// TIA Portal V20 export
DATA_BLOCK "InstStackCalculateDB"   // DB459
// stored: InstanceOfName 2201_StackCalculate, InstanceOfType FB
"2201_StackCalculate"
   // VAR_INPUT
   //    Execute : Bool;
   //    Direction : Bool;
   //    CPM : LReal;
   //    StageWidth : LReal;
   //    StageHeight : LReal;
   //    StageGap : LReal;
   //    AccRatio : DInt;
   //    RatioOption : Bool;
   //    TimeOption : Bool;
   //    PosOption : Bool;
   //    DoubleOption : Bool;
   //    Ratio : Struct
   //       FinalRollerStart : LReal;
   //       FinalRollerEnd : LReal;
   //       PnPXStart : LReal;
   //       PnPXEnd : LReal;
   //       PnPZDownStart : LReal;
   //       PnPZDownEnd : LReal;
   //       PnPZUpStart : LReal;
   //       PnPZUpEnd : LReal;
   //       MandrelBwdStart : LReal;
   //       MandrelBwdEnd : LReal;
   //       MandrelFwdStart : LReal;
   //       MandrelFwdEnd : LReal;
   //       MandrelUpStart1 : LReal;
   //       MandrelUpEnd1 : LReal;
   //       MandrelUpStart2 : LReal;
   //       MandrelUpEnd2 : LReal;
   //       MandrelDownStart : LReal;
   //       MandrelDownEnd : LReal;
   //       MandrelYTerm : LReal;
   //       MandrelZTerm : LReal;
   //       MandrelBwdOffset : LReal;
   //       MandrelFwdOffset : LReal;
   //    END_STRUCT;
   //    "Time" : Struct
   //       FinalRollerStart : LReal;
   //       FinalRollerEnd : LReal;
   //       PnPXStart : LReal;
   //       PnPXEnd : LReal;
   //       PnPZDownStart : LReal;
   //       PnPZDownEnd : LReal;
   //       PnPZUpStart : LReal;
   //       PnPZUpEnd : LReal;
   //       MandrelBwdStart : LReal;
   //       MandrelBwdEnd : LReal;
   //       MandrelFwdStart : LReal;
   //       MandrelFwdEnd : LReal;
   //       MandrelUpStart1 : LReal;
   //       MandrelUpEnd1 : LReal;
   //       MandrelUpStart2 : LReal;
   //       MandrelUpEnd2 : LReal;
   //       MandrelDownStart : LReal;
   //       MandrelDownEnd : LReal;
   //    END_STRUCT;
   //    Position : Struct
   //       FinalRollerBwdPos : LReal;
   //       FinalRollerFwdPos : LReal;
   //    END_STRUCT;
   //    FinalRollerDistance : LReal;
   //    AnodePnPX1Distance : LReal;
   //    AnodePnPX2Distance : LReal;
   //    CathodePnPX1Distance : LReal;
   //    CathodePnPX2Distance : LReal;
   //    AnodePnPZ1Distance1 : LReal;
   //    AnodePnPZ1Distance2 : LReal;
   //    AnodePnPZ2Distance1 : LReal;
   //    AnodePnPZ2Distance2 : LReal;
   //    CathodePnPZ1Distance1 : LReal;
   //    CathodePnPZ1Distance2 : LReal;
   //    CathodePnPZ2Distance1 : LReal;
   //    CathodePnPZ2Distance2 : LReal;
   //    AnodeMandrelYFrontDistance : LReal;
   //    AnodeMandrelYRearDistance : LReal;
   //    CathodeMandrelYFrontDistance : LReal;
   //    CathodeMandrelYRearDistance : LReal;
   //    AnodeMandrelZFrontDistance : LReal;
   //    AnodeMandrelZRearDistance : LReal;
   //    CathodeMandrelZFrontDistance : LReal;
   //    CathodeMandrelZRearDistance : LReal;
   // END_VAR
   // VAR_OUTPUT
   //    Done : Bool;
   //    Busy : Bool;
   //    Error : Bool;
   //    ErrorID : DWord;
   //    StatusID : DWord;
   //    NowCmd : DInt;
   //    BeforeCmd : DInt;
   // END_VAR
   // VAR_IN_OUT
   //    EmptyPoint : Array[1..10000] of TO_Cam_Struct_PointData;
   //    EmptySegment : Array[1..50] of TO_Cam_Struct_SegmentData;
   //    FinalRollerCam : DB_ANY;
   //    CompensatorCam : DB_ANY;
   //    AnodePnPX1Cam : DB_ANY;
   //    AnodePnPX2Cam : DB_ANY;
   //    AnodePnPZ1Cam : DB_ANY;
   //    AnodePnPZ2Cam : DB_ANY;
   //    CathodePnPX1Cam : DB_ANY;
   //    CathodePnPX2Cam : DB_ANY;
   //    CathodePnPZ1Cam : DB_ANY;
   //    CathodePnPZ2Cam : DB_ANY;
   //    AnodeMandrelYFrontCam : DB_ANY;
   //    AnodeMandrelYRearCam : DB_ANY;
   //    AnodeMandrelZFrontCam : DB_ANY;
   //    AnodeMandrelZRearCam : DB_ANY;
   //    CathodeMandrelYFrontCam : DB_ANY;
   //    CathodeMandrelYRearCam : DB_ANY;
   //    CathodeMandrelZFrontCam : DB_ANY;
   //    CathodeMandrelZRearCam : DB_ANY;
   // END_VAR
   // VAR
   //    statNowCmd : DInt;
   //    statBeforeCmd : DInt;
   //    statLineSpeed : LReal;
   //    statTargetBwdTime : LReal;
   //    statTargetFwdTime : LReal;
   //    statTimeTable : Array[1..50] of Time;
   //    statStartTime : Time;
   //    statEndTime : Time;
   //    instTriggerExecute : R_TRIG;
   //    instCalculateFinalRoller { S7_SetPoint := 'True'} : "2303_CalculateCam_FinalRoller";
   //    instCalculateBwdTime { S7_SetPoint := 'True'} : "2304_CalculateCam_FinalTime";
   //    instCalculateFwdTime { S7_SetPoint := 'True'} : "2304_CalculateCam_FinalTime";
   //    instCalculateCompensator { S7_SetPoint := 'True'} : "2305_CalculateCam_Compensator";
   //    instCalculateAnodePnPX1 { S7_SetPoint := 'True'} : "2301_CalculateCam_PnPX";
   //    instCalculateAnodePnPX2 { S7_SetPoint := 'True'} : "2301_CalculateCam_PnPX";
   //    instCalculateAnodePnPZ1 { S7_SetPoint := 'True'} : "2302_CalculateCam_PnPZ";
   //    instCalculateAnodePnPZ2 { S7_SetPoint := 'True'} : "2302_CalculateCam_PnPZ";
   //    instCalculateCathodePnPX1 { S7_SetPoint := 'True'} : "2301_CalculateCam_PnPX";
   //    instCalculateCathodePnPX2 { S7_SetPoint := 'True'} : "2301_CalculateCam_PnPX";
   //    instCalculateCathodePnPZ1 { S7_SetPoint := 'True'} : "2302_CalculateCam_PnPZ";
   //    instCalculateCathodePnPZ2 { S7_SetPoint := 'True'} : "2302_CalculateCam_PnPZ";
   //    instCalculateMandrelYFront1 { S7_SetPoint := 'True'} : "2307_CalculateCam_MandrelY1";
   //    instCalculateMandrelYRear1 { S7_SetPoint := 'True'} : "2307_CalculateCam_MandrelY1";
   //    instCalculateMandrelZFront1 { S7_SetPoint := 'True'} : "2306_CalculateCam_MandrelZ1";
   //    instCalculateMandrelZRear1 { S7_SetPoint := 'True'} : "2306_CalculateCam_MandrelZ1";
   //    instCalculateMandrelYFront2 { S7_SetPoint := 'True'} : "2309_CalculateCam_MandrelY2";
   //    instCalculateMandrelYRear2 { S7_SetPoint := 'True'} : "2309_CalculateCam_MandrelY2";
   //    instCalculateMandrelZFront2 { S7_SetPoint := 'True'} : "2308_CalculateCam_MandrelZ2";
   //    instCalculateMandrelZRear2 { S7_SetPoint := 'True'} : "2308_CalculateCam_MandrelZ2";
   // END_VAR
BEGIN
END_DATA_BLOCK
